METHOD FB_init : BOOL
VAR_INPUT
  /// if TRUE, the retain variables are initialized (warm start / cold start)
  bInitRetains : BOOL; 
  /// if TRUE, the instance afterwards gets moved into the copy code (online change)
  bInCopyCode  : BOOL;  
END_VAR
MyType := 'MC_CalculateInverseKinematicFB';

ExecMode := ExecutionMode.PARALLEL;
END_METHOD

METHOD PROTECTED OnCall
VAR_IN_OUT
  /// Robot assignment of function
  AxesGroup : AxesGroup; 
END_VAR
// call base implementation
SUPER^.OnCall(AxesGroup := AxesGroup);

CASE _stepCmd OF
  
  00:  IF ( _execute_R.Q )  
       THEN
         // Check function is supported and parameter are valid ?
         IF (( CheckFunctionSupported( AxesGroup := AxesGroup )) AND
             ( CheckParameterValid   ( AxesGroup := AxesGroup )))      
         THEN
           // set busy flag
           Busy := TRUE;
           // Reset command outputs
           SysDepMemSet(pDest := ADR(OutCmd), Value := 0, DataLen := SIZEOF(OutCmd));         
           // apply command parameter
          _parCmd := ParCmd;
           // init parameter sequence
          _command.ParSeq := 1;
           // create command data
           CommandData := CreateCommandPayload(AxesGroup := AxesGroup);
           // Add command to active command register
          _uniqueID := AxesGroup.Acyclic.ActiveCommandRegister.AddCmd( pCommandFB := ADR(THIS^ ));     
           // set timeout
           SetTimeout(PT := _timeoutCmd, rTimer := _timerCmd);
           // inc step counter
          _stepCmd := _stepCmd + 1;
         END_IF 
       END_IF
     

  01:  // Wait for responce received
       IF ( _responseReceived )
       THEN
         // reset response received flag
        _responseReceived := FALSE;

         CASE  _response.State 
         OF
           CmdMessageState.BUFFERED : CommandBuffered := TRUE;
           CmdMessageState.DONE     : Done            := TRUE;
           CmdMessageState.ERROR    : Error           := TRUE;
         END_CASE
                
         // Done, Aborted or Error ?
         IF (_response.State >= CmdMessageState.DONE )
         THEN
           // Reset Busy flag
           Busy := FALSE;
           // Update results
           OutCmd.JointPosition := _response.JointPosition;
           // set timeout
           SetTimeout(PT := _timeoutCmd, rTimer := _timerCmd);
           // inc step counter
          _stepCmd := _stepCmd + 1; 
         END_IF
       END_IF


  02: IF ( NOT Execute)
      THEN
        Reset();
      END_IF     

ELSE
  // invalid step
  ErrorID := RobotLibraryEvents.ERR_INVALID_STEP;
END_CASE


// Reset FB
IF ( NOT Execute )
THEN
  Reset();
END_IF
END_METHOD

METHOD INTERNAL ParseResponsePayload : DINT
VAR_INPUT
  /// Response data
  ResponseData : RobotLibraryRecvDataFB;
  /// Timestamp
  Timestamp    : SystemTime;  
END_VAR
// Table 6-639: Received CMD payload (RC to PLC) of "CalculateInverseKinematic"
// --------------------------
// Header
// --------------------------
// Byte 00 : USINT - ParSeq | State     
// Byte 01 : SINT  - AlarmMessageSeverity    
// Byte 02 : UINT  - AlarmMessageCode HB
// Byte 03 :       - AlarmMessageCode LB
// --------------------------
// Datablock
// --------------------------
// Byte 04 : REAL  - JointPosition.J1  HW HB
// Byte 05 :       - JointPosition.J1  HW LB
// Byte 06 :       - JointPosition.J1  LW HB
// Byte 07 :       - JointPosition.J1  LW LB
// Byte 08 : REAL  - JointPosition.J2  HW HB
// Byte 09 :       - JointPosition.J2 HW LB
// Byte 10 :       - JointPosition.J2  LW HB
// Byte 11 :       - JointPosition.J2  LW LB
// Byte 12 : REAL  - JointPosition.J3  HW HB
// Byte 13 :       - JointPosition.J3  HW LB
// Byte 14 :       - JointPosition.J3  LW HB
// Byte 15 :       - JointPosition.J3  LW LB
// Byte 16 : REAL  - JointPosition.J4  HW HB
// Byte 17 :       - JointPosition.J4  HW LB
// Byte 18 :       - JointPosition.J4  LW HB
// Byte 19 :       - JointPosition.J4  LW LB
// Byte 20 : REAL  - JointPosition.J5  HW HB
// Byte 21 :       - JointPosition.J5  HW LB
// Byte 22 :       - JointPosition.J5  LW HB
// Byte 23 :       - JointPosition.J5  LW LB
// Byte 24 : REAL  - JointPosition.J6  HW HB
// Byte 25 :       - JointPosition.J6  HW LB
// Byte 26 :       - JointPosition.J6  LW HB
// Byte 27 :       - JointPosition.J6  LW LB
// Byte 28 : REAL  - JointPosition.E1  HW HB
// Byte 29 :       - JointPosition.E1  HW LB
// Byte 30 :       - JointPosition.E1  LW HB
// Byte 31 :       - JointPosition.E1  LW LB
// Byte 32 : REAL  - JointPosition.E2  HW HB
// Byte 33 :       - JointPosition.E2  HW LB
// Byte 34 :       - JointPosition.E2  LW HB
// Byte 35 :       - JointPosition.E2  LW LB
// Byte 36 : REAL  - JointPosition.E3  HW HB
// Byte 37 :       - JointPosition.E3  HW LB
// Byte 38 :       - JointPosition.E3  LW HB
// Byte 39 :       - JointPosition.E3  LW LB
// Byte 40 : REAL  - JointPosition.E4  HW HB
// Byte 41 :       - JointPosition.E4  HW LB
// Byte 42 :       - JointPosition.E4  LW HB
// Byte 43 :       - JointPosition.E4  LW LB
// Byte 44 : REAL  - JointPosition.E5  HW HB
// Byte 45 :       - JointPosition.E5  HW LB
// Byte 46 :       - JointPosition.E5  LW HB
// Byte 47 :       - JointPosition.E5  LW LB
// Byte 48 : REAL  - JointPosition.E6  HW HB
// Byte 49 :       - JointPosition.E6  HW LB
// Byte 50 :       - JointPosition.E6  LW HB
// Byte 51 :       - JointPosition.E6  LW LB
// --------------------------
// call base implementation to parse the header from payload buffer
ResponseData.PayloadPtr := SUPER^.ParseResponsePayload(ResponseData := ResponseData, Timestamp := Timestamp);

// copy parsed header to response
_response.ParSeq               := _rspHeader.ParSeq;
_response.State                := _rspHeader.State;
_response.AlarmMessageSeverity := _rspHeader.AlarmMessageSeverity;
_response.AlarmMessageCode     := _rspHeader.AlarmMessageCode;

// Get Response.JointPosition.J1
_response.JointPosition.J1 := ResponseData.GetReal();
// Get Response.JointPosition.J2
_response.JointPosition.J2 := ResponseData.GetReal();
// Get Response.JointPosition.J3
_response.JointPosition.J3 := ResponseData.GetReal();
// Get Response.JointPosition.J4
_response.JointPosition.J4 := ResponseData.GetReal();
// Get Response.JointPosition.J5
_response.JointPosition.J5 := ResponseData.GetReal();
// Get Response.JointPosition.J6
_response.JointPosition.J6 := ResponseData.GetReal();
// Get Response.JointPosition.E1
_response.JointPosition.E1 := ResponseData.GetReal();
// Get Response.JointPosition.E2
_response.JointPosition.E2 := ResponseData.GetReal();
// Get Response.JointPosition.E3
_response.JointPosition.E3 := ResponseData.GetReal();
// Get Response.JointPosition.E4
_response.JointPosition.E4 := ResponseData.GetReal();
// Get Response.JointPosition.E5
_response.JointPosition.E5 := ResponseData.GetReal();
// Get Response.JointPosition.E6
_response.JointPosition.E6 := ResponseData.GetReal();

// Create logging
ParseResponsePayloadLog(ResponseData := ResponseData, Timestamp := Timestamp);
END_METHOD

METHOD INTERNAL ParseResponsePayloadLog
VAR_INPUT
  /// Response data
  ResponseData : RobotLibraryRecvDataFB;
  /// Timestamp
  Timestamp    : SystemTime;  
END_VAR
// Create log entry for Parameter start
CreateLogMessage      ( Timestamp   := Timestamp,
                        MessageType := MessageType.CMD,
                        Severity    := Severity.DEBUG,
                        MessageCode := 0,
                        MessageText := 'Parsed the following parameter(s) from response data:');
                        
// Create log entry for JointPosition.J1
CreateLogMessagePara1 ( Timestamp   := Timestamp,
                        MessageType := MessageType.CMD,
                        Severity    := Severity.DEBUG,
                        MessageCode := 0,
                        MessageText := 'Response.JointPosition.J1 = {1}',
                        Para1       :=  REAL_TO_STRING(_response.JointPosition.J1));

// Create log entry for JointPosition.J2
CreateLogMessagePara1 ( Timestamp   := Timestamp,
                        MessageType := MessageType.CMD,
                        Severity    := Severity.DEBUG,
                        MessageCode := 0,
                        MessageText := 'Response.JointPosition.J2 = {1}',
                        Para1       :=  REAL_TO_STRING(_response.JointPosition.J2));

// Create log entry for JointPosition.J3
CreateLogMessagePara1 ( Timestamp   := Timestamp,
                        MessageType := MessageType.CMD,
                        Severity    := Severity.DEBUG,
                        MessageCode := 0,
                        MessageText := 'Response.JointPosition.J3 = {1}',
                        Para1       :=  REAL_TO_STRING(_response.JointPosition.J3));

// Create log entry for JointPosition.J4
CreateLogMessagePara1 ( Timestamp   := Timestamp,
                        MessageType := MessageType.CMD,
                        Severity    := Severity.DEBUG,
                        MessageCode := 0,
                        MessageText := 'Response.JointPosition.J4 = {1}',
                        Para1       :=  REAL_TO_STRING(_response.JointPosition.J4));

// Create log entry for JointPosition.J5
CreateLogMessagePara1 ( Timestamp   := Timestamp,
                        MessageType := MessageType.CMD,
                        Severity    := Severity.DEBUG,
                        MessageCode := 0,
                        MessageText := 'Response.JointPosition.J5 = {1}',
                        Para1       :=  REAL_TO_STRING(_response.JointPosition.J5));

// Create log entry for JointPosition.J6
CreateLogMessagePara1 ( Timestamp   := Timestamp,
                        MessageType := MessageType.CMD,
                        Severity    := Severity.DEBUG,
                        MessageCode := 0,
                        MessageText := 'Response.JointPosition.J6 = {1}',
                        Para1       :=  REAL_TO_STRING(_response.JointPosition.J6));

// Create log entry for JointPosition.E1
CreateLogMessagePara1 ( Timestamp   := Timestamp,
                        MessageType := MessageType.CMD,
                        Severity    := Severity.DEBUG,
                        MessageCode := 0,
                        MessageText := 'Response.JointPosition.E1 = {1}',
                        Para1       :=  REAL_TO_STRING(_response.JointPosition.E1));

// Create log entry for JointPosition.E2
CreateLogMessagePara1 ( Timestamp   := Timestamp,
                        MessageType := MessageType.CMD,
                        Severity    := Severity.DEBUG,
                        MessageCode := 0,
                        MessageText := 'Response.JointPosition.E2 = {1}',
                        Para1       :=  REAL_TO_STRING(_response.JointPosition.E2));

// Create log entry for JointPosition.E3
CreateLogMessagePara1 ( Timestamp   := Timestamp,
                        MessageType := MessageType.CMD,
                        Severity    := Severity.DEBUG,
                        MessageCode := 0,
                        MessageText := 'Response.JointPosition.E3 = {1}',
                        Para1       :=  REAL_TO_STRING(_response.JointPosition.E3));

// Create log entry for JointPosition.E4
CreateLogMessagePara1 ( Timestamp   := Timestamp,
                        MessageType := MessageType.CMD,
                        Severity    := Severity.DEBUG,
                        MessageCode := 0,
                        MessageText := 'Response.JointPosition.E4 = {1}',
                        Para1       :=  REAL_TO_STRING(_response.JointPosition.E4));

// Create log entry for JointPosition.E5
CreateLogMessagePara1 ( Timestamp   := Timestamp,
                        MessageType := MessageType.CMD,
                        Severity    := Severity.DEBUG,
                        MessageCode := 0,
                        MessageText := 'Response.JointPosition.E5 = {1}',
                        Para1       :=  REAL_TO_STRING(_response.JointPosition.E5));

// Create log entry for JointPosition.E6
CreateLogMessagePara1 ( Timestamp   := Timestamp,
                        MessageType := MessageType.CMD,
                        Severity    := Severity.DEBUG,
                        MessageCode := 0,
                        MessageText := 'Response.JointPosition.E6 = {1}',
                        Para1       :=  REAL_TO_STRING(_response.JointPosition.E6));
END_METHOD

METHOD PROTECTED Reset : DINT
VAR_INPUT
END_VAR
Reset := SUPER^.Reset();

Done               := FALSE;
Busy               := FALSE;
CommandBuffered    := FALSE;
END_METHOD

END_FUNCTION_BLOCK

// Library/POUs/Calculation/MC_CalculateTool/MC_CalculateToolFB
/// Calculate tool (TCP) with four-point method
FUNCTION_BLOCK MC_CalculateToolFB EXTENDS RobotLibraryBaseExecuteFB
// ------------------------------------------------------------------------- 
//  SRCI Robot Library                                                
// ------------------------------------------------------------------------- 
//                                                                           
//  Object:      CalculateToolFB                                       
//  Author:      Thorsten Brach                                                
//  Date:        2024-06-09
//
//  Description:                                              
//   
//                                                                           
//  Copyright: 
//    (C) 2024 Thorsten Brach. All rights reserved                                                                                                                                            
//             Licensed under the LGPL-3.0 license.
//                                                                           
//  Disclaimer:                                                                           
//    This project is provided without any guarantee and can be used for   
//    private and commercial purposes. Any use is at the user’s 
//    own risk and responsibility.
//
// -------------------------------------------------------------------------
VAR_INPUT
  /// Command parameter 
  ParCmd          : CalculateToolParCmd;      
END_VAR
VAR_OUTPUT
  /// Command is transferred and confirmed by the RC
  CommandBuffered : BOOL;
  /// Command output 
  OutCmd          : CalculateToolOutCmd;  
END_VAR

VAR
  /// internal copy of command parameter 
 _parCmd          : CalculateToolParCmd;
  /// command data to send
 _command         : CalculateToolSendData;
  /// response data received
 _response        : CalculateToolRecvData;      
  /// Incremented with each position of the input parameter "PositionsArray" sent from the PLC to the RC.
  /// • Default: 0
 _dataIndex       : USINT;
  /// Set TRUE by the client, when according to the user selected "Mode" the final position of the input parameter "PositionsArray" is sent to the RC.
  /// • Default: FALSE
 _dataComplete    : BOOL;
END_VAR

SUPER^(AxesGroup := AxesGroup);

METHOD PROTECTED CheckFunctionSupported : BOOL
VAR_IN_OUT
  /// Robot assignment of function
  AxesGroup : AxesGroup; 
END_VAR
CheckFunctionSupported := AxesGroup.InternalData.RCSupportedFunctions.CalculateTool;

IF ( NOT CheckFunctionSupported )
THEN
  // call base implementation for set error and create log entry
  SUPER^.CheckFunctionSupported(AxesGroup := AxesGroup);
END_IF
END_METHOD

METHOD PROTECTED CheckParameterChanged : BOOL
VAR_IN_OUT
  /// Robot assignment of function
  AxesGroup    : AxesGroup; 
END_VAR
// Check ParCmd Size is > 0, because MemCmp does not work correctly with size = 0
IF (SIZEOF(ParCmd) = 0) 
THEN 
  RETURN;
END_IF

// compare memory 
_parameterChanged := ( SysDepMemCmp(pData1 := ADR(ParCmd), pData2 := ADR(_parCmd), DataLen := SIZEOF(ParCmd)) <> RobotLibraryConstants.OK );

// check parameter valid ?
_parameterValid   := CheckParameterValid( AxesGroup := AxesGroup );

IF ((  _parameterChanged        )  AND 
    (  _parameterValid          )) OR
    (  _parameterUpdateInternal )  
THEN  
  // reset internal flag for send parameter update
 _parameterUpdateInternal := FALSE;
  // update internal copy of parameters 
 _parCmd := ParCmd;
  // inc parameter sequence
 _command.ParSeq := _command.ParSeq + 1;
  // update command data  
  CommandData := CreateCommandPayload(AxesGroup := AxesGroup); // ( Access via reference to rCommandFB in ACR )
  // notify active command register 
  AxesGroup.Acyclic.ActiveCommandRegister.NotifyParameterChanged := _uniqueID;
END_IF
END_METHOD

METHOD INTERNAL CreateCommandPayload : RobotLibrarySendDataFB
VAR_IN_OUT
  /// Robot assignment of function
  AxesGroup : AxesGroup; 
END_VAR
// Table 6-650: Sent CMD payload (PLC to RC) of "CalculateTool"
// --------------------------
// Header
// --------------------------
// Byte 00 : UINT       - Type HB     
// Byte 01 :            - Type LB    
// Byte 02 : USINT      - Reserve | ExecutionMode
// Byte 03 : USINT      - ParSeq  | Priority
// --------------------------
// Datablock
// --------------------------
// Byte 04 : USINT      - DataIndex
// Byte 05 : BOOL       - DataComplete
// Byte 06 : USINT      - ToolNo
// Byte 07 : USINT      - FrameNo
// Byte 08 : SINT       - Mode
// Byte 09 : USINT      - ExternalTCP
// Byte 10 : REAL       - Position.X  HW HB
// Byte 11 :            - Position.X  HW LB
// Byte 12 :            - Position.X  LW HB
// Byte 13 :            - Position.X  LW LB
// Byte 14 : REAL       - Position.Y  HW HB
// Byte 15 :            - Position.Y  HW LB
// Byte 16 :            - Position.Y  LW HB
// Byte 17 :            - Position.Y  LW LB
// Byte 18 : REAL       - Position.Z  HW HB
// Byte 19 :            - Position.Z  HW LB
// Byte 20 :            - Position.Z  LW HB
// Byte 21 :            - Position.Z  LW LB
// Byte 22 : REAL       - Position.Rx HW HB
// Byte 23 :            - Position.Rx HW LB
// Byte 24 :            - Position.Rx LW HB
// Byte 25 :            - Position.Rx LW LB
// Byte 26 : REAL       - Position.Ry HW HB
// Byte 27 :            - Position.Ry HW LB
// Byte 28 :            - Position.Ry LW HB
// Byte 29 :            - Position.Ry LW LB
// Byte 30 : REAL       - Position.Rz HW HB
// Byte 31 :            - Position.Rz HW LB
// Byte 32 :            - Position.Rz LW HB
// Byte 33 :            - Position.Rz LW LB
// Byte 34 : Config     - ArmConfig   LW HB
// Byte 35 :            - ArmConfig   LW LB
// Byte 36 : TurnNumber - J1 + J2     LW HB
// Byte 37 :            - J3 + J4     LW LB
// Byte 38 :            - J5 + J6     LW LB
// Byte 39 :            - E1          LW LB
// Byte 40 : REAL       - Position.E1 HW HB
// Byte 41 :            - Position.E1 HW LB
// Byte 42 :            - Position.E1 LW HB
// Byte 43 :            - Position.E1 LW LB
// Byte 44 : REAL       - Position.E2 HW HB
// Byte 45 :            - Position.E2 HW LB
// Byte 46 :            - Position.E2 LW HB
// Byte 47 :            - Position.E2 LW LB
// Byte 48 : REAL       - Position.E3 HW HB
// Byte 49 :            - Position.E3 HW LB
// Byte 50 :            - Position.E3 LW HB
// Byte 51 :            - Position.E3 LW LB
// Byte 52 : REAL       - Position.E4 HW HB
// Byte 53 :            - Position.E4 HW LB
// Byte 54 :            - Position.E4 LW HB
// Byte 55 :            - Position.E4 LW LB
// Byte 56 : REAL       - Position.E5 HW HB
// Byte 57 :            - Position.E5 HW LB
// Byte 58 :            - Position.E5 LW HB
// Byte 59 :            - Position.E5 LW LB
// Byte 60 : REAL       - Position.E6 HW HB
// Byte 61 :            - Position.E6 HW LB
// Byte 62 :            - Position.E6 LW HB
// Byte 63 :            - Position.E6 LW LB
// --------------------------
// set command parameter 
_command.CmdTyp         :=  CmdType.CalculateTool;
_command.ExecMode       :=  ExecMode;
_command.ParSeq         := _command.ParSeq;
_command.Priority       :=  Priority;
_command.DataIndex      := _dataIndex;
_command.DataComplete.0 := _dataComplete;
_command.ToolNo         := _parCmd.ToolNo;
_command.FrameNo        := _parCmd.FrameNo;
_command.Mode           := _parCmd.Mode;
_command.ExternalTCP.0  := _parCmd.ExternalTCP;
  
// copy command data to header
_cmdHeader := _command;
// call base implementation to copy header to payload buffer
CreateCommandPayload := SUPER^.CreateCommandPayload(AxesGroup := AxesGroup);

// add command.TargetFrameNo
CreateCommandPayload.AddUsint(_command.DataIndex);
// add command.DataComplete
CreateCommandPayload.AddByte(_command.DataComplete);
// add command.ToolNo
CreateCommandPayload.AddUsint(_command.ToolNo);
// add command.FrameNo
CreateCommandPayload.AddUsint(_command.FrameNo);
// add command.Mode
CreateCommandPayload.AddSint(_command.Mode);
// add command.Mode
CreateCommandPayload.AddUsint(_command.ExternalTCP);
// add command.Position.X
CreateCommandPayload.AddReal(_command.Position.X);
// add command.Position.Y
CreateCommandPayload.AddReal(_command.Position.Y);
// add command.Position.Z
CreateCommandPayload.AddReal(_command.Position.Z);
// add command.Position.Rx
CreateCommandPayload.AddReal(_command.Position.Rx);
// add command.Position.Ry
CreateCommandPayload.AddReal(_command.Position.Ry);
// add command.Position.Rz
CreateCommandPayload.AddReal(_command.Position.Rz);
// add command.Position.Config
CreateCommandPayload.AddArmConfig (_command.Position.Config);
// add command.Position.TurnNumber
CreateCommandPayload.AddTurnNumber(_command.Position.TurnNumber);
// add command.Position.E1
CreateCommandPayload.AddReal(_command.Position.E1);
// add command.Position.E2
CreateCommandPayload.AddReal(_command.Position.E2);
// add command.Position.E3
CreateCommandPayload.AddReal(_command.Position.E3);
// add command.Position.E4
CreateCommandPayload.AddReal(_command.Position.E4);
// add command.Position.E5
CreateCommandPayload.AddReal(_command.Position.E5);
// add command.Position.E6
CreateCommandPayload.AddReal(_command.Position.E6);

// Create logging
CreateCommandPayloadLog(AxesGroup := AxesGroup);
END_METHOD

METHOD INTERNAL CreateCommandPayloadLog 
VAR_IN_OUT
  /// Robot assignment of function
  AxesGroup : AxesGroup; 
END_VAR
// Create log entry for Parameter start
CreateLogMessage      ( Timestamp   := AxesGroup.InternalData.SystemTime,
                        MessageType := MessageType.CMD,
                        Severity    := Severity.DEBUG,
                        MessageCode := 0,
                        MessageText := 'Create command payload with the following parameter(s) :');

// Create log entry for DataIndex
CreateLogMessagePara1 ( Timestamp   := AxesGroup.InternalData.SystemTime,
                        MessageType := MessageType.CMD,
                        Severity    := Severity.DEBUG,
                        MessageCode := 0,
                        MessageText := 'Command.DataIndex = {1}',
                        Para1       :=  USINT_TO_STRING(_command.DataIndex));

// Create log entry for DataComplete
CreateLogMessagePara1 ( Timestamp   := AxesGroup.InternalData.SystemTime,
                        MessageType := MessageType.CMD,
                        Severity    := Severity.DEBUG,
                        MessageCode := 0,
                        MessageText := 'Command.DataComplete = {1}',
                        Para1       :=  BYTE_TO_STRING(_command.DataComplete));

// Create log entry for ToolNo
CreateLogMessagePara1 ( Timestamp   := AxesGroup.InternalData.SystemTime,
                        MessageType := MessageType.CMD,
                        Severity    := Severity.DEBUG,
                        MessageCode := 0,
                        MessageText := 'Command.ToolNo = {1}',
                        Para1       :=  USINT_TO_STRING(_command.ToolNo));

// Create log entry for FrameNo
CreateLogMessagePara1 ( Timestamp   := AxesGroup.InternalData.SystemTime,
                        MessageType := MessageType.CMD,
                        Severity    := Severity.DEBUG,
                        MessageCode := 0,
                        MessageText := 'Command.FrameNo = {1}',
                        Para1       :=  USINT_TO_STRING(_command.FrameNo));

// Create log entry for Mode
CreateLogMessagePara1 ( Timestamp   := AxesGroup.InternalData.SystemTime,
                        MessageType := MessageType.CMD,
                        Severity    := Severity.DEBUG,
                        MessageCode := 0,
                        MessageText := 'Command.Mode = {1}',
                        Para1       :=  TOOL_CALCULATION_MODE_TO_STRING(_command.Mode));

// Create log entry for ExternalTCP
CreateLogMessagePara1 ( Timestamp   := AxesGroup.InternalData.SystemTime,
                        MessageType := MessageType.CMD,
                        Severity    := Severity.DEBUG,
                        MessageCode := 0,
                        MessageText := 'Command.ExternalTCP = {1}',
                        Para1       :=  BOOL_TO_STRING(_command.ExternalTCP.0));

// Create log entry for Position.X
CreateLogMessagePara1 ( Timestamp   := AxesGroup.InternalData.SystemTime,
                        MessageType := MessageType.CMD,
                        Severity    := Severity.DEBUG,
                        MessageCode := 0,
                        MessageText := 'Command.Position.X = {1}',
                        Para1       :=  REAL_TO_STRING(_command.Position.X));

// Create log entry for Position.Y
CreateLogMessagePara1 ( Timestamp   := AxesGroup.InternalData.SystemTime,
                        MessageType := MessageType.CMD,
                        Severity    := Severity.DEBUG,
                        MessageCode := 0,
                        MessageText := 'Command.Position.Y = {1}',
                        Para1       :=  REAL_TO_STRING(_command.Position.Y));

// Create log entry for Position.Z
CreateLogMessagePara1 ( Timestamp   := AxesGroup.InternalData.SystemTime,
                        MessageType := MessageType.CMD,
                        Severity    := Severity.DEBUG,
                        MessageCode := 0,
                        MessageText := 'Command.Position.Z = {1}',
                        Para1       :=  REAL_TO_STRING(_command.Position.Z));

// Create log entry for Position.Rx
CreateLogMessagePara1 ( Timestamp   := AxesGroup.InternalData.SystemTime,
                        MessageType := MessageType.CMD,
                        Severity    := Severity.DEBUG,
                        MessageCode := 0,
                        MessageText := 'Command.Position.Rx = {1}',
                        Para1       :=  REAL_TO_STRING(_command.Position.Rx));

// Create log entry for Position.Ry
CreateLogMessagePara1 ( Timestamp   := AxesGroup.InternalData.SystemTime,
                        MessageType := MessageType.CMD,
                        Severity    := Severity.DEBUG,
                        MessageCode := 0,
                        MessageText := 'Command.Position.Ry = {1}',
                        Para1       :=  REAL_TO_STRING(_command.Position.Ry));

// Create log entry for Position.Rz
CreateLogMessagePara1 ( Timestamp   := AxesGroup.InternalData.SystemTime,
                        MessageType := MessageType.CMD,
                        Severity    := Severity.DEBUG,
                        MessageCode := 0,
                        MessageText := 'Command.Position.Rz = {1}',
                        Para1       :=  REAL_TO_STRING(_command.Position.Rz));

// Create log entry for Position.Config
CreateLogMessagePara1 ( Timestamp   := AxesGroup.InternalData.SystemTime,
                        MessageType := MessageType.CMD,
                        Severity    := Severity.DEBUG,
                        MessageCode := 0,
                        MessageText := 'Command.Position.Config = {1}',
                        Para1       :=  ARM_CONFIG_TO_STRING(_command.Position.Config));

// Create log entry for Position.TurnNumber[0]
CreateLogMessagePara1 ( Timestamp   := AxesGroup.InternalData.SystemTime,
                        MessageType := MessageType.CMD,
                        Severity    := Severity.DEBUG,
                        MessageCode := 0,
                        MessageText := 'Command.Position.TurnNumber[0] = {1}',
                        Para1       :=  BYTE_TO_STRING(CombineHalfSints(HalfSintHi := _command.Position.TurnNumber.J2Turns, 
                                                                        HalfSintLo := _command.Position.TurnNumber.J1Turns)));

// Create log entry for Position.TurnNumber[1]
CreateLogMessagePara1 ( Timestamp   := AxesGroup.InternalData.SystemTime,
                        MessageType := MessageType.CMD,
                        Severity    := Severity.DEBUG,
                        MessageCode := 0,
                        MessageText := 'Command.Position.TurnNumber[1] = {1}',
                        Para1       :=  BYTE_TO_STRING(CombineHalfSints(HalfSintHi := _command.Position.TurnNumber.J4Turns, 
                                                                        HalfSintLo := _command.Position.TurnNumber.J3Turns)));

// Create log entry for Position.TurnNumber[2]
CreateLogMessagePara1 ( Timestamp   := AxesGroup.InternalData.SystemTime,
                        MessageType := MessageType.CMD,
                        Severity    := Severity.DEBUG,
                        MessageCode := 0,
                        MessageText := 'Command.Position.TurnNumber[2] = {1}',
                        Para1       :=  BYTE_TO_STRING(CombineHalfSints(HalfSintHi := _command.Position.TurnNumber.J6Turns, 
                                                                        HalfSintLo := _command.Position.TurnNumber.J5Turns)));

// Create log entry for Position.TurnNumber[3]
CreateLogMessagePara1 ( Timestamp   := AxesGroup.InternalData.SystemTime,
                        MessageType := MessageType.CMD,
                        Severity    := Severity.DEBUG,
                        MessageCode := 0,
                        MessageText := 'Command.Position.TurnNumber[3] = {1}',
                        Para1       :=  SINT_TO_STRING(_command.Position.TurnNumber.E1Turns));

// Create log entry for Position.E1
CreateLogMessagePara1 ( Timestamp   := AxesGroup.InternalData.SystemTime,
                        MessageType := MessageType.CMD,
                        Severity    := Severity.DEBUG,
                        MessageCode := 0,
                        MessageText := 'Command.Position.E1 = {1}',
                        Para1       :=  REAL_TO_STRING(_command.Position.E1));

// Create log entry for Position.E2
CreateLogMessagePara1 ( Timestamp   := AxesGroup.InternalData.SystemTime,
                        MessageType := MessageType.CMD,
                        Severity    := Severity.DEBUG,
                        MessageCode := 0,
                        MessageText := 'Command.Position.E2 = {1}',
                        Para1       :=  REAL_TO_STRING(_command.Position.E2));

// Create log entry for Position.E3
CreateLogMessagePara1 ( Timestamp   := AxesGroup.InternalData.SystemTime,
                        MessageType := MessageType.CMD,
                        Severity    := Severity.DEBUG,
                        MessageCode := 0,
                        MessageText := 'Command.Position.E3 = {1}',
                        Para1       :=  REAL_TO_STRING(_command.Position.E3));

// Create log entry for Position.E4
CreateLogMessagePara1 ( Timestamp   := AxesGroup.InternalData.SystemTime,
                        MessageType := MessageType.CMD,
                        Severity    := Severity.DEBUG,
                        MessageCode := 0,
                        MessageText := 'Command.Position.E4 = {1}',
                        Para1       :=  REAL_TO_STRING(_command.Position.E4));

// Create log entry for Position.E5
CreateLogMessagePara1 ( Timestamp   := AxesGroup.InternalData.SystemTime,
                        MessageType := MessageType.CMD,
                        Severity    := Severity.DEBUG,
                        MessageCode := 0,
                        MessageText := 'Command.Position.E5 = {1}',
                        Para1       :=  REAL_TO_STRING(_command.Position.E5));

// Create log entry for Position.E6
CreateLogMessagePara1 ( Timestamp   := AxesGroup.InternalData.SystemTime,
                        MessageType := MessageType.CMD,
                        Severity    := Severity.DEBUG,
                        MessageCode := 0,
                        MessageText := 'Command.Position.E6 = {1}',
                        Para1       :=  REAL_TO_STRING(_command.Position.E6));
END_METHOD

METHOD FB_init : BOOL
VAR_INPUT
  /// if TRUE, the retain variables are initialized (warm start / cold start)
  bInitRetains : BOOL; 
  /// if TRUE, the instance afterwards gets moved into the copy code (online change)
  bInCopyCode  : BOOL;  
END_VAR
MyType := 'MC_CalculateToolFB';

ExecMode := ExecutionMode.PARALLEL;
END_METHOD

METHOD PROTECTED OnCall
VAR_IN_OUT
  /// Robot assignment of function
  AxesGroup : AxesGroup; 
END_VAR
// call base implementation
SUPER^.OnCall(AxesGroup := AxesGroup);

CASE _stepCmd OF
  
  00:  IF ( _execute_R.Q )  
       THEN
         // Check function is supported and parameter are valid ?
         IF (( CheckFunctionSupported( AxesGroup := AxesGroup )) AND
             ( CheckParameterValid   ( AxesGroup := AxesGroup )))      
         THEN
           // set busy flag
           Busy := TRUE;
           // Reset command outputs
           SysDepMemSet(pDest := ADR(OutCmd), Value := 0, DataLen := SIZEOF(OutCmd));         
           // apply command parameter
          _parCmd := ParCmd;
           // init parameter sequence
          _command.ParSeq := 1;
           // set timeout
           SetTimeout(PT := _timeoutCmd, rTimer := _timerCmd);
           // inc step counter
          _stepCmd := _stepCmd + 1;
         END_IF 
       END_IF
     

  01: // inc data index 
     _dataIndex := _dataIndex + 1;

      CASE _parCmd.Mode OF

        ToolCalculationMode.TWO_POINT_Z_METHOD :
          _dataComplete := _dataIndex >= 2;
        
        ToolCalculationMode.THREE_POINT_METHOD :
          _dataComplete := _dataIndex >= 3;

        ToolCalculationMode.FOUR_POINT_METHOD :
          _dataComplete := _dataIndex >= 4;        

        ToolCalculationMode.FIVE_POINT_METHOD :        
          _dataComplete := _dataIndex >= 5;

        ToolCalculationMode.SIX_POINT_METHOD :        
          _dataComplete := _dataIndex >= 6;

        ToolCalculationMode.ABC_WORLD_METHOD :
          _dataComplete := _dataIndex >= 1;
        
        ToolCalculationMode.ABC_TWO_POINT_METHOD :
          _dataComplete := _dataIndex >= 2;

      END_CASE

       // create command data
       CommandData := CreateCommandPayload(AxesGroup := AxesGroup);
       // Add command to active command register
      _uniqueID := AxesGroup.Acyclic.ActiveCommandRegister.AddCmd( pCommandFB := ADR(THIS^ ));     
       // set timeout
       SetTimeout(PT := _timeoutCmd, rTimer := _timerCmd);
       // inc step counter
      _stepCmd := _stepCmd + 1; 


  02:  // Wait for responce received
       IF ( _responseReceived )
       THEN
         // reset response received flag
        _responseReceived := FALSE;

         CASE  _response.State 
         OF
           CmdMessageState.BUFFERED : CommandBuffered := TRUE;
           CmdMessageState.DONE     : Done            := TRUE;
           CmdMessageState.ERROR    : Error           := TRUE;
         END_CASE
                
         // Done, Aborted or Error ?
         IF (_response.State >= CmdMessageState.DONE )
         THEN
           // Reset Busy flag
           Busy := FALSE;
           // Update results
           OutCmd.TCPMaxError    := _response.TCPMaxError;
           OutCmd.TCPMeanError   := _response.TCPMeanError;
           OutCmd.ToolData       := _response.ToolData;
           
           IF ( _dataComplete ) OR (_response.State = CmdMessageState.ABORTED )
           THEN
             // set timeout
             SetTimeout(PT := _timeoutCmd, rTimer := _timerCmd);
             // inc step counter
            _stepCmd := _stepCmd + 1; 
           ELSE
             // set timeout
             SetTimeout(PT := _timeoutCmd, rTimer := _timerCmd);
             // dec step counter
            _stepCmd := _stepCmd - 1; 
           END_IF
         END_IF
       END_IF


  03: IF ( NOT Execute)
      THEN
        Reset(); 
      END_IF     
      
ELSE
  // invalid step
  ErrorID := RobotLibraryEvents.ERR_INVALID_STEP;
END_CASE


// Reset FB
IF ( NOT Execute )
THEN
  Reset();
END_IF
END_METHOD

METHOD INTERNAL ParseResponsePayload : DINT
VAR_INPUT
  /// Response data
  ResponseData : RobotLibraryRecvDataFB;
  /// Timestamp
  Timestamp    : SystemTime;  
END_VAR
// Table 6-651: Received CMD payload (RC to PLC) of "CalculateTool"
// --------------------------
// Header
// --------------------------
// Byte 00 : USINT      - ParSeq | State     
// Byte 01 : SINT       - AlarmMessageSeverity    
// Byte 02 : UINT       - AlarmMessageCode HB
// Byte 03 :            - AlarmMessageCode LB
// --------------------------
// Datablock
// --------------------------
// Byte 04 : IEC_DATE   - ToolData.Date LW HB
// Byte 05 :            - ToolData.Date LW LB
// Byte 06 : REAL       - TCPMaxError   HW HB
// Byte 07 :            - TCPMaxError   HW LB
// Byte 08 :            - TCPMaxError   LW HB
// Byte 09 :            - TCPMaxError   LW LB
// Byte 10 : REAL       - TCPMeanError  HW HB
// Byte 11 :            - TCPMeanError  HW LB
// Byte 12 :            - TCPMeanError  LW HB
// Byte 13 :            - TCPMeanError  LW LB
// Byte 14 : IEC_TIME   - ToolData.Time HW HB
// Byte 15 :            - ToolData.Time HW LB
// Byte 16 :            - ToolData.Time LW HB
// Byte 17 :            - ToolData.Time LW LB


// Byte 18 : REAL       - ToolData.X  HW HB
// Byte 19 :            - ToolData.X  HW LB
// Byte 20 :            - ToolData.X  LW HB
// Byte 21 :            - ToolData.X  LW LB
// Byte 22 : REAL       - ToolData.Y  HW HB
// Byte 23 :            - ToolData.Y  HW LB
// Byte 24 :            - ToolData.Y  LW HB
// Byte 25 :            - ToolData.Y  LW LB
// Byte 26 : REAL       - ToolData.Z  HW HB
// Byte 27 :            - ToolData.Z  HW LB
// Byte 28 :            - ToolData.Z  LW HB
// Byte 29 :            - ToolData.Z  LW LB
// Byte 30 : REAL       - ToolData.Rx HW HB
// Byte 31 :            - ToolData.Rx HW LB
// Byte 32 :            - ToolData.Rx LW HB
// Byte 33 :            - ToolData.Rx LW LB
// Byte 34 : REAL       - ToolData.Ry HW HB
// Byte 35 :            - ToolData.Ry HW LB
// Byte 36 :            - ToolData.Ry LW HB
// Byte 37 :            - ToolData.Ry LW LB
// Byte 38 : REAL       - ToolData.Rz HW HB
// Byte 39 :            - ToolData.Rz HW LB
// Byte 40 :            - ToolData.Rz LW HB
// Byte 41 :            - ToolData.Rz LW LB
// Byte 42 : USINT      - ToolData.ID
// Byte 43 : USINT      - ToolData.LoadNo
// Byte 44 : BOOL       - ToolData.ExternalTCP
// --------------------------
// call base implementation to parse the header from payload buffer
ResponseData.PayloadPtr := SUPER^.ParseResponsePayload(ResponseData := ResponseData, Timestamp := Timestamp);

// copy parsed header to response
_response.ParSeq                := _rspHeader.ParSeq;
_response.State                 := _rspHeader.State;
_response.AlarmMessageSeverity  := _rspHeader.AlarmMessageSeverity;
_response.AlarmMessageCode      := _rspHeader.AlarmMessageCode;

// Get Response.IEC_Date
_response.ToolData.Timestamp.IEC_Date := ResponseData.GetIecDate();
// Get Response.TCPMaxError
_response.TCPMaxError := ResponseData.GetReal();
// Get Response.TCPMeanError
_response.TCPMeanError := ResponseData.GetReal();
// Get Response.ToolData.Time
_response.ToolData.Timestamp.IEC_Time := ResponseData.GetIecTime();
// Get Response.ToolData.X
_response.ToolData.X := ResponseData.GetReal();
// Get Response.ToolData.Y            
_response.ToolData.Y := ResponseData.GetReal();
// Get Response.ToolData.Z            
_response.ToolData.Z := ResponseData.GetReal();
// Get Response.ToolData.Rx           
_response.ToolData.Rx := ResponseData.GetReal();
// Get Response.ToolData.Ry           
_response.ToolData.Ry := ResponseData.GetReal();
// Get Response.ToolData.Rz           
_response.ToolData.Rz := ResponseData.GetReal();
// Get Response.ToolData.ID           
_response.ToolData.ID := ResponseData.GetUsint();
// Get Response.ToolData.LoadNo       
_response.ToolData.LoadNo := ResponseData.GetUsint();
// Get Response.ToolData.ExternalTCP
_response.ToolData.ExternalTCP := ResponseData.GetBool();

// Create logging
ParseResponsePayloadLog(ResponseData := ResponseData, Timestamp := Timestamp);
END_METHOD

METHOD INTERNAL ParseResponsePayloadLog
VAR_INPUT
  /// Response data
  ResponseData : RobotLibraryRecvDataFB;
  /// Timestamp
  Timestamp    : SystemTime;  
END_VAR
// Create log entry for Parameter start
CreateLogMessage      ( Timestamp   := Timestamp,
                        MessageType := MessageType.CMD,
                        Severity    := Severity.DEBUG,
                        MessageCode := 0,
                        MessageText := 'Parsed the following parameter(s) from response data:');
                        
// Create log entry for IEC_Date
CreateLogMessagePara1 ( Timestamp   := Timestamp,
                        MessageType := MessageType.CMD,
                        Severity    := Severity.DEBUG,
                        MessageCode := 0,
                        MessageText := 'Response.ToolData.Timestamp.IEC_DATE = {1}',
                        Para1       :=  IEC_DATE_TO_STRING(_response.ToolData.Timestamp.IEC_DATE));

// Create log entry for TCPMaxError
CreateLogMessagePara1 ( Timestamp   := Timestamp,
                        MessageType := MessageType.CMD,
                        Severity    := Severity.DEBUG,
                        MessageCode := 0,
                        MessageText := 'Response.TCPMaxError = {1}',
                        Para1       :=  REAL_TO_STRING(_response.TCPMaxError));

// Create log entry for TCPMeanError
CreateLogMessagePara1 ( Timestamp   := Timestamp,
                        MessageType := MessageType.CMD,
                        Severity    := Severity.DEBUG,
                        MessageCode := 0,
                        MessageText := 'Response.TCPMeanError = {1}',
                        Para1       :=  REAL_TO_STRING(_response.TCPMeanError));

// Create log entry for IEC_Time
CreateLogMessagePara1 ( Timestamp   := Timestamp,
                        MessageType := MessageType.CMD,
                        Severity    := Severity.DEBUG,
                        MessageCode := 0,
                        MessageText := 'Response.ToolData.Timestamp.IEC_TIME = {1}',
                        Para1       :=  IEC_TIME_TO_STRING(_response.ToolData.Timestamp.IEC_TIME));

// Create log entry for ToolData.X
CreateLogMessagePara1 ( Timestamp   := Timestamp,
                        MessageType := MessageType.CMD,
                        Severity    := Severity.DEBUG,
                        MessageCode := 0,
                        MessageText := 'Response.ToolData.X = {1}',
                        Para1       :=  REAL_TO_STRING(_response.ToolData.X));

// Create log entry for ToolData.Y
CreateLogMessagePara1 ( Timestamp   := Timestamp,
                        MessageType := MessageType.CMD,
                        Severity    := Severity.DEBUG,
                        MessageCode := 0,
                        MessageText := 'Response.ToolData.Y = {1}',
                        Para1       :=  REAL_TO_STRING(_response.ToolData.Y));

// Create log entry for ToolData.Z
CreateLogMessagePara1 ( Timestamp   := Timestamp,
                        MessageType := MessageType.CMD,
                        Severity    := Severity.DEBUG,
                        MessageCode := 0,
                        MessageText := 'Response.ToolData.Z = {1}',
                        Para1       :=  REAL_TO_STRING(_response.ToolData.Z));

// Create log entry for ToolData.Rx
CreateLogMessagePara1 ( Timestamp   := Timestamp,
                        MessageType := MessageType.CMD,
                        Severity    := Severity.DEBUG,
                        MessageCode := 0,
                        MessageText := 'Response.ToolData.Rx = {1}',
                        Para1       :=  REAL_TO_STRING(_response.ToolData.Rx));

// Create log entry for ToolData.Ry
CreateLogMessagePara1 ( Timestamp   := Timestamp,
                        MessageType := MessageType.CMD,
                        Severity    := Severity.DEBUG,
                        MessageCode := 0,
                        MessageText := 'Response.ToolData.Ry = {1}',
                        Para1       :=  REAL_TO_STRING(_response.ToolData.Ry));

// Create log entry for ToolData.Rz
CreateLogMessagePara1 ( Timestamp   := Timestamp,
                        MessageType := MessageType.CMD,
                        Severity    := Severity.DEBUG,
                        MessageCode := 0,
                        MessageText := 'Response.ToolData.Rz = {1}',
                        Para1       :=  REAL_TO_STRING(_response.ToolData.Rz));

// Create log entry for ToolData.ID
CreateLogMessagePara1 ( Timestamp   := Timestamp,
                        MessageType := MessageType.CMD,
                        Severity    := Severity.DEBUG,
                        MessageCode := 0,
                        MessageText := 'Response.ToolData.ID = {1}',
                        Para1       :=  USINT_TO_STRING(_response.ToolData.ID));

// Create log entry for ToolData.LoadNo
CreateLogMessagePara1 ( Timestamp   := Timestamp,
                        MessageType := MessageType.CMD,
                        Severity    := Severity.DEBUG,
                        MessageCode := 0,
                        MessageText := 'Response.ToolData.LoadNo = {1}',
                        Para1       :=  USINT_TO_STRING(_response.ToolData.LoadNo));

// Create log entry for ToolData.ExternalTCP
CreateLogMessagePara1 ( Timestamp   := Timestamp,
                        MessageType := MessageType.CMD,
                        Severity    := Severity.DEBUG,
                        MessageCode := 0,
                        MessageText := 'Response.ToolData.ExternalTCP = {1}',
                        Para1       :=  BOOL_TO_STRING(_response.ToolData.ExternalTCP));
END_METHOD

METHOD PROTECTED Reset : DINT
VAR_INPUT
END_VAR
Reset := SUPER^.Reset();

Done               := FALSE;
Busy               := FALSE;
CommandBuffered    := FALSE;
END_METHOD

END_FUNCTION_BLOCK

// Library/POUs/Calculation/MC_LoadMeasurementAutomatic/MC_LoadMeasurementAutomaticFB
/// Automatic detection of load data
FUNCTION_BLOCK MC_LoadMeasurementAutomaticFB EXTENDS RobotLibraryBaseExecuteFB
// ------------------------------------------------------------------------- 
//  SRCI Robot Library                                                
// ------------------------------------------------------------------------- 
//                                                                           
//  Object:      LoadMeasurementAutomaticFB                                       
//  Author:      Thorsten Brach                                                
//  Date:        2024-06-01
//
//  Description:                                              
//   
//                                                                           
//  Copyright: 
//    (C) 2024 Thorsten Brach. All rights reserved                                                                                                                                            
//             Licensed under the LGPL-3.0 license.
//                                                                           
//  Disclaimer:                                                                           
//    This project is provided without any guarantee and can be used for   
//    private and commercial purposes. Any use is at the user’s 
//    own risk and responsibility.
//
// -------------------------------------------------------------------------
VAR_INPUT
  /// Parameter which determines the behavior towards the previously sent and still active or buffered commands.
  AbortingMode    : AbortingMode;
  /// Defines the target sequence in which the command will be executed
  SequenceFlag    : SequenceFlag;  
  /// Command parameter 
  ParCmd          : LoadMeasurementAutomaticParCmd;      
END_VAR

VAR_OUTPUT
  /// Command is transferred and confirmed by the RC
  CommandBuffered    : BOOL;  
  /// The command takes control of the motion of the according axis group.
  Active             : BOOL;
  /// The command was aborted by another command.
  CommandAborted     : BOOL;
  /// TRUE, while command is interrupted during execution and can be continued.
  CommandInterrupted : BOOL;
  /// Command output 
  OutCmd             : LoadMeasurementAutomaticOutCmd;        
END_VAR

VAR
  /// internal copy of command parameter 
 _parCmd          : LoadMeasurementAutomaticParCmd;
  /// command data to send
 _command         : LoadMeasurementAutomaticSendData;
  /// response data received
 _response        : LoadMeasurementAutomaticRecvData;      
END_VAR

SUPER^(AxesGroup := AxesGroup);

METHOD PROTECTED CheckFunctionSupported : BOOL
VAR_IN_OUT
  /// Robot assignment of function
  AxesGroup : AxesGroup; 
END_VAR
CheckFunctionSupported := AxesGroup.InternalData.RCSupportedFunctions.LoadMeasurementAutomatic;

IF ( NOT CheckFunctionSupported )
THEN
  // call base implementation for set error and create log entry
  SUPER^.CheckFunctionSupported(AxesGroup := AxesGroup);
END_IF
END_METHOD

METHOD PROTECTED CheckParameterChanged : BOOL
VAR_IN_OUT
  /// Robot assignment of function
  AxesGroup    : AxesGroup; 
END_VAR
// Check ParCmd Size is > 0, because MemCmp does not work correctly with size = 0
IF (SIZEOF(ParCmd) = 0) 
THEN 
  RETURN;
END_IF

// compare memory 
_parameterChanged := ( SysDepMemCmp(pData1 := ADR(ParCmd), pData2 := ADR(_parCmd), DataLen := SIZEOF(ParCmd)) <> RobotLibraryConstants.OK );

// check parameter valid ?
_parameterValid   := CheckParameterValid( AxesGroup := AxesGroup );

IF ((  _parameterChanged        )  AND 
    (  _parameterValid          )) OR
    (  _parameterUpdateInternal )  
THEN  
  // reset internal flag for send parameter update
 _parameterUpdateInternal := FALSE;
  // update internal copy of parameters 
 _parCmd := ParCmd;
  // inc parameter sequence
 _command.ParSeq := _command.ParSeq + 1;
  // update command data  
  CommandData := CreateCommandPayload(AxesGroup := AxesGroup); // ( Access via reference to rCommandFB in ACR )
  // notify active command register 
  AxesGroup.Acyclic.ActiveCommandRegister.NotifyParameterChanged := _uniqueID;
END_IF
END_METHOD

METHOD INTERNAL CreateCommandPayload : RobotLibrarySendDataFB
VAR_IN_OUT
  /// Robot assignment of function
  AxesGroup : AxesGroup; 
END_VAR
// Table 6-778: Sent CMD payload (PLC to RC) of "LoadMeasurementAutomatic"
// --------------------------
// Header
// --------------------------
// Byte 000 : UINT  - Type HB     
// Byte 001 :       - Type LB    
// Byte 002 : USINT - Reserve | ExecutionMode
// Byte 003 : USINT - ParSeq  | Priority
// --------------------------
// Datablock
// --------------------------
// Byte 004 : REAL       - Mass HW HB
// Byte 005 :            - Mass HW LB
// Byte 006 :            - Mass LW HB
// Byte 007 :            - Mass LW LB
// Byte 008 : USINT      - Mode
// Byte 009 : BYTE       - Reserved
// Byte 010 : REAL       - AreaJ3[0] HW HB
// Byte 011 :            - AreaJ3[0] HW LB
// Byte 012 :            - AreaJ3[0] LW HB
// Byte 013 :            - AreaJ3[0] LW LB
// Byte 014 : REAL       - AreaJ3[1] HW HB
// Byte 015 :            - AreaJ3[1] HW LB
// Byte 016 :            - AreaJ3[1] LW HB
// Byte 017 :            - AreaJ3[1] LW LB
// Byte 018 : REAL       - AreaJ4[0] HW HB
// Byte 019 :            - AreaJ4[0] HW LB
// Byte 020 :            - AreaJ4[0] LW HB
// Byte 021 :            - AreaJ4[0] LW LB
// Byte 022 : REAL       - AreaJ4[1] HW HB
// Byte 023 :            - AreaJ4[1] HW LB
// Byte 024 :            - AreaJ4[1] LW HB
// Byte 025 :            - AreaJ4[1] LW LB
// Byte 026 : REAL       - AreaJ5[0] HW HB
// Byte 027 :            - AreaJ5[0] HW LB
// Byte 028 :            - AreaJ5[0] LW HB
// Byte 029 :            - AreaJ5[0] LW LB
// Byte 030 : REAL       - AreaJ5[1] HW HB
// Byte 031 :            - AreaJ5[1] HW LB
// Byte 032 :            - AreaJ5[1] LW HB
// Byte 033 :            - AreaJ5[1] LW LB
// Byte 034 : REAL       - AreaJ6[0] HW HB
// Byte 035 :            - AreaJ6[0] HW LB
// Byte 036 :            - AreaJ6[0] LW HB
// Byte 037 :            - AreaJ6[0] LW LB
// Byte 038 : REAL       - AreaJ6[1] HW HB
// Byte 039 :            - AreaJ6[1] HW LB
// Byte 040 :            - AreaJ6[1] LW HB
// Byte 041 :            - AreaJ6[1] LW LB
// Byte 042 : REAL       - ConfigurationAngle HW HB
// Byte 043 :            - ConfigurationAngle HW LB
// Byte 044 :            - ConfigurationAngle LW HB
// Byte 045 :            - ConfigurationAngle LW LB
// Byte 046 : REAL       - Position_1.J1 HW HB
// Byte 047 :            - Position_1.J1 HW LB
// Byte 048 :            - Position_1.J1 LW HB
// Byte 049 :            - Position_1.J1 LW LB
// Byte 050 : REAL       - Position_1.J2 HW HB
// Byte 051 :            - Position_1.J2 HW LB
// Byte 052 :            - Position_1.J2 LW HB
// Byte 053 :            - Position_1.J2 LW LB
// Byte 054 : REAL       - Position_1.J3 HW HB
// Byte 055 :            - Position_1.J3 HW LB
// Byte 056 :            - Position_1.J3 LW HB
// Byte 057 :            - Position_1.J3 LW LB
// Byte 058 : REAL       - Position_1.J4 HW HB
// Byte 059 :            - Position_1.J4 HW LB
// Byte 060 :            - Position_1.J4 LW HB
// Byte 061 :            - Position_1.J4 LW LB
// Byte 062 : REAL       - Position_1.J5 HW HB
// Byte 063 :            - Position_1.J5 HW LB
// Byte 064 :            - Position_1.J5 LW HB
// Byte 065 :            - Position_1.J5 LW LB
// Byte 066 : REAL       - Position_1.J6 HW HB
// Byte 067 :            - Position_1.J6 HW LB
// Byte 068 :            - Position_1.J6 LW HB
// Byte 069 :            - Position_1.J6 LW LB
// Byte 070 : REAL       - Position_1.E1 HW HB
// Byte 071 :            - Position_1.E1 HW LB
// Byte 072 :            - Position_1.E1 LW HB
// Byte 073 :            - Position_1.E1 LW LB
// Byte 074 : REAL       - Position_2.J1 HW HB
// Byte 075 :            - Position_2.J1 HW LB
// Byte 076 :            - Position_2.J1 LW HB
// Byte 077 :            - Position_2.J1 LW LB
// Byte 078 : REAL       - Position_2.J2 HW HB
// Byte 079 :            - Position_2.J2 HW LB
// Byte 080 :            - Position_2.J2 LW HB
// Byte 081 :            - Position_2.J2 LW LB
// Byte 082 : REAL       - Position_2.J3 HW HB
// Byte 083 :            - Position_2.J3 HW LB
// Byte 084 :            - Position_2.J3 LW HB
// Byte 085 :            - Position_2.J3 LW LB
// Byte 086 : REAL       - Position_2.J4 HW HB
// Byte 087 :            - Position_2.J4 HW LB
// Byte 088 :            - Position_2.J4 LW HB
// Byte 089 :            - Position_2.J4 LW LB
// Byte 090 : REAL       - Position_2.J5 HW HB
// Byte 091 :            - Position_2.J5 HW LB
// Byte 092 :            - Position_2.J5 LW HB
// Byte 093 :            - Position_2.J5 LW LB
// Byte 094 : REAL       - Position_2.J6 HW HB
// Byte 095 :            - Position_2.J6 HW LB
// Byte 096 :            - Position_2.J6 LW HB
// Byte 097 :            - Position_2.J6 LW LB
// Byte 098 : REAL       - Position_2.E1 HW HB
// Byte 099 :            - Position_2.E1 HW LB
// Byte 100 :            - Position_2.E1 LW HB
// Byte 101 :            - Position_2.E1 LW LB
// Byte 102 : REAL       - Position_1.E1 HW HB
// Byte 103 :            - Position_1.E2 HW LB
// Byte 104 :            - Position_1.E2 LW HB
// Byte 105 :            - Position_1.E2 LW LB
// Byte 106 : REAL       - Position_1.E3 HW HB
// Byte 107 :            - Position_1.E3 HW LB
// Byte 108 :            - Position_1.E3 LW HB
// Byte 109 :            - Position_1.E3 LW LB
// Byte 110 : REAL       - Position_1.E4 HW HB
// Byte 111 :            - Position_1.E4 HW LB
// Byte 112 :            - Position_1.E4 LW HB
// Byte 113 :            - Position_1.E4 LW LB
// Byte 114 : REAL       - Position_1.E5 HW HB
// Byte 115 :            - Position_1.E5 HW LB
// Byte 116 :            - Position_1.E5 LW HB
// Byte 117 :            - Position_1.E5 LW LB
// Byte 118 : REAL       - Position_1.E6 HW HB
// Byte 119 :            - Position_1.E6 HW LB
// Byte 120 :            - Position_1.E6 LW HB
// Byte 121 :            - Position_1.E6 LW LB
// Byte 122 : REAL       - Position_2.E2 HW HB
// Byte 123 :            - Position_2.E2 HW LB
// Byte 124 :            - Position_2.E2 LW HB
// Byte 125 :            - Position_2.E2 LW LB
// Byte 125 : REAL       - Position_2.E3 HW HB
// Byte 127 :            - Position_2.E3 HW LB
// Byte 128 :            - Position_2.E3 LW HB
// Byte 129 :            - Position_2.E3 LW LB
// Byte 130 : REAL       - Position_2.E4 HW HB
// Byte 131 :            - Position_2.E4 HW LB
// Byte 132 :            - Position_2.E4 LW HB
// Byte 133 :            - Position_2.E4 LW LB
// Byte 134 : REAL       - Position_2.E5 HW HB
// Byte 135 :            - Position_2.E5 HW LB
// Byte 136 :            - Position_2.E5 LW HB
// Byte 137 :            - Position_2.E5 LW LB
// Byte 138 : REAL       - Position_2.E6 HW HB
// Byte 139 :            - Position_2.E6 HW LB
// Byte 140 :            - Position_2.E6 LW HB
// Byte 141 :            - Position_2.E6 LW LB
// set command parameter 
_command.CmdTyp             :=  CmdType.LoadMeasurementAutomatic;
_command.ExecMode           :=  ExecMode;
_command.ParSeq             := _command.ParSeq;
_command.Priority           :=  Priority;

_command.Mass               := parCmd.Mass;
_command.Mode               := parCmd.Mode;
_command.Reserved           := 0;
_command.Area_J3            := parCmd.Area_J3;
_command.Area_J4            := parCmd.Area_J4;
_command.Area_J5            := parCmd.Area_J5;
_command.Area_J6            := parCmd.Area_J6;
_command.ConfigurationAngle := parCmd.ConfigurationAngle;
_command.Position_1         := parCmd.Position_1;
_command.Position_2         := parCmd.Position_2;


// copy command data to header
_cmdHeader := _command;
// call base implementation to copy header to payload buffer
CreateCommandPayload := SUPER^.CreateCommandPayload(AxesGroup := AxesGroup);

// add command.Mass
CreateCommandPayload.AddReal(_command.Mass);
// add command.Mode
CreateCommandPayload.AddUsint(_command.Mode);
// add command.Reserved
CreateCommandPayload.AddByte(_command.Reserved);
// add command.Area_J3[0]
CreateCommandPayload.AddReal(_command.Area_J3[0]);
// add command.Area_J3[1]
CreateCommandPayload.AddReal(_command.Area_J3[1]);
// add command.Area_J4[0]
CreateCommandPayload.AddReal(_command.Area_J4[0]);
// add command.Area_J4[1]
CreateCommandPayload.AddReal(_command.Area_J4[1]);
// add command.Area_J5[0]
CreateCommandPayload.AddReal(_command.Area_J5[0]);
// add command.Area_J5[1]
CreateCommandPayload.AddReal(_command.Area_J5[1]);
// add command.Area_J6[0]
CreateCommandPayload.AddReal(_command.Area_J6[0]);
// add command.Area_J6[1]
CreateCommandPayload.AddReal(_command.Area_J6[1]);
// add command.ConfigurationAngle
CreateCommandPayload.AddReal(_command.ConfigurationAngle);
// add command.Position_1.J1
CreateCommandPayload.AddReal(_command.Position_1.J1);
// add command.Position_1.J2
CreateCommandPayload.AddReal(_command.Position_1.J2);
// add command.Position_1.J3
CreateCommandPayload.AddReal(_command.Position_1.J3);
// add command.Position_1.J4
CreateCommandPayload.AddReal(_command.Position_1.J4);
// add command.Position_1.J5
CreateCommandPayload.AddReal(_command.Position_1.J5);
// add command.Position_1.J6
CreateCommandPayload.AddReal(_command.Position_1.J6);
// add command.Position_1.E1
CreateCommandPayload.AddReal(_command.Position_1.E1);
// add command.Position_1.E2
CreateCommandPayload.AddReal(_command.Position_1.E2);
// add command.Position_1.E3
CreateCommandPayload.AddReal(_command.Position_1.E3);
// add command.Position_1.E4
CreateCommandPayload.AddReal(_command.Position_1.E4);
// add command.Position_1.E5
CreateCommandPayload.AddReal(_command.Position_1.E5);
// add command.Position_1.E6
CreateCommandPayload.AddReal(_command.Position_1.E6);
// add command.Position_2.J1
CreateCommandPayload.AddReal(_command.Position_2.J1);
// add command.Position_2.J2
CreateCommandPayload.AddReal(_command.Position_2.J2);
// add command.Position_2.J3
CreateCommandPayload.AddReal(_command.Position_2.J3);
// add command.Position_2.J4
CreateCommandPayload.AddReal(_command.Position_2.J4);
// add command.Position_2.J5
CreateCommandPayload.AddReal(_command.Position_2.J5);
// add command.Position_2.J6
CreateCommandPayload.AddReal(_command.Position_2.J6);
// add command.Position_2.E1
CreateCommandPayload.AddReal(_command.Position_2.E1);
// add command.Position_2.E2
CreateCommandPayload.AddReal(_command.Position_2.E2);
// add command.Position_2.E3
CreateCommandPayload.AddReal(_command.Position_2.E3);
// add command.Position_2.E4
CreateCommandPayload.AddReal(_command.Position_2.E4);
// add command.Position_2.E5
CreateCommandPayload.AddReal(_command.Position_2.E5);
// add command.Position_2.E6
CreateCommandPayload.AddReal(_command.Position_2.E6);

// Create logging
CreateCommandPayloadLog(AxesGroup := AxesGroup);
END_METHOD

METHOD INTERNAL CreateCommandPayloadLog 
VAR_IN_OUT
  /// Robot assignment of function
  AxesGroup : AxesGroup; 
END_VAR
// Create log entry for Parameter start
CreateLogMessage      ( Timestamp   := AxesGroup.InternalData.SystemTime,
                        MessageType := MessageType.CMD,
                        Severity    := Severity.DEBUG,
                        MessageCode := 0,
                        MessageText := 'Create command payload with the following parameter(s) :');

// Create log entry for Mass
CreateLogMessagePara1 ( Timestamp   := AxesGroup.InternalData.SystemTime,
                        MessageType := MessageType.CMD,
                        Severity    := Severity.DEBUG,
                        MessageCode := 0,
                        MessageText := 'Command.Mass = {1}',
                        Para1       :=  REAL_TO_STRING(_command.Mass));

// Create log entry for Mode
CreateLogMessagePara1 ( Timestamp   := AxesGroup.InternalData.SystemTime,
                        MessageType := MessageType.CMD,
                        Severity    := Severity.DEBUG,
                        MessageCode := 0,
                        MessageText := 'Command.Mode = {1}',
                        Para1       :=  LOAD_MEASUREMENT_MODE_TO_STRING(_command.Mode));

// Create log entry for Reserved
CreateLogMessagePara1 ( Timestamp   := AxesGroup.InternalData.SystemTime,
                        MessageType := MessageType.CMD,
                        Severity    := Severity.DEBUG,
                        MessageCode := 0,
                        MessageText := 'Command.Reserved = {1}',
                        Para1       :=  REAL_TO_STRING(_command.Reserved));

// Create log entry for Area_J3[0]
CreateLogMessagePara1 ( Timestamp   := AxesGroup.InternalData.SystemTime,
                        MessageType := MessageType.CMD,
                        Severity    := Severity.DEBUG,
                        MessageCode := 0,
                        MessageText := 'Command.Area_J3[0] = {1}',
                        Para1       :=  REAL_TO_STRING(_command.Area_J3[0]));

// Create log entry for Area_J3[1]
CreateLogMessagePara1 ( Timestamp   := AxesGroup.InternalData.SystemTime,
                        MessageType := MessageType.CMD,
                        Severity    := Severity.DEBUG,
                        MessageCode := 0,
                        MessageText := 'Command.Area_J3[1] = {1}',
                        Para1       :=  REAL_TO_STRING(_command.Area_J3[1]));
                        
// Create log entry for Area_J4[0]
CreateLogMessagePara1 ( Timestamp   := AxesGroup.InternalData.SystemTime,
                        MessageType := MessageType.CMD,
                        Severity    := Severity.DEBUG,
                        MessageCode := 0,
                        MessageText := 'Command.Area_J4[0] = {1}',
                        Para1       :=  REAL_TO_STRING(_command.Area_J4[0]));

// Create log entry for Area_J4[1]
CreateLogMessagePara1 ( Timestamp   := AxesGroup.InternalData.SystemTime,
                        MessageType := MessageType.CMD,
                        Severity    := Severity.DEBUG,
                        MessageCode := 0,
                        MessageText := 'Command.Area_J4[1] = {1}',
                        Para1       :=  REAL_TO_STRING(_command.Area_J4[1]));

// Create log entry for Area_J5[0]
CreateLogMessagePara1 ( Timestamp   := AxesGroup.InternalData.SystemTime,
                        MessageType := MessageType.CMD,
                        Severity    := Severity.DEBUG,
                        MessageCode := 0,
                        MessageText := 'Command.Area_J5[0] = {1}',
                        Para1       :=  REAL_TO_STRING(_command.Area_J5[0]));

// Create log entry for Area_J5[1]
CreateLogMessagePara1 ( Timestamp   := AxesGroup.InternalData.SystemTime,
                        MessageType := MessageType.CMD,
                        Severity    := Severity.DEBUG,
                        MessageCode := 0,
                        MessageText := 'Command.Area_J5[1] = {1}',
                        Para1       :=  REAL_TO_STRING(_command.Area_J5[1]));
                        
// Create log entry for Area_J6[0]
CreateLogMessagePara1 ( Timestamp   := AxesGroup.InternalData.SystemTime,
                        MessageType := MessageType.CMD,
                        Severity    := Severity.DEBUG,
                        MessageCode := 0,
                        MessageText := 'Command.Area_J6[0] = {1}',
                        Para1       :=  REAL_TO_STRING(_command.Area_J6[0]));

// Create log entry for Area_J6[1]
CreateLogMessagePara1 ( Timestamp   := AxesGroup.InternalData.SystemTime,
                        MessageType := MessageType.CMD,
                        Severity    := Severity.DEBUG,
                        MessageCode := 0,
                        MessageText := 'Command.Area_J6[1] = {1}',
                        Para1       :=  REAL_TO_STRING(_command.Area_J6[1]));
                        
// Create log entry for ConfigurationAngle
CreateLogMessagePara1 ( Timestamp   := AxesGroup.InternalData.SystemTime,
                        MessageType := MessageType.CMD,
                        Severity    := Severity.DEBUG,
                        MessageCode := 0,
                        MessageText := 'Command.ConfigurationAngle = {1}',
                        Para1       :=  REAL_TO_STRING(_command.ConfigurationAngle));

// Create log entry for Position_1.J1
CreateLogMessagePara1 ( Timestamp   := AxesGroup.InternalData.SystemTime,
                        MessageType := MessageType.CMD,
                        Severity    := Severity.DEBUG,
                        MessageCode := 0,
                        MessageText := 'Command.Position_1.J1 = {1}',
                        Para1       :=  REAL_TO_STRING(_command.Position_1.J1));

// Create log entry for Position_1.J2
CreateLogMessagePara1 ( Timestamp   := AxesGroup.InternalData.SystemTime,
                        MessageType := MessageType.CMD,
                        Severity    := Severity.DEBUG,
                        MessageCode := 0,
                        MessageText := 'Command.Position_1.J2 = {1}',
                        Para1       :=  REAL_TO_STRING(_command.Position_1.J2));
                        
// Create log entry for Position_1.J3
CreateLogMessagePara1 ( Timestamp   := AxesGroup.InternalData.SystemTime,
                        MessageType := MessageType.CMD,
                        Severity    := Severity.DEBUG,
                        MessageCode := 0,
                        MessageText := 'Command.Position_1.J3 = {1}',
                        Para1       :=  REAL_TO_STRING(_command.Position_1.J3));
                        
// Create log entry for Position_1.J4
CreateLogMessagePara1 ( Timestamp   := AxesGroup.InternalData.SystemTime,
                        MessageType := MessageType.CMD,
                        Severity    := Severity.DEBUG,
                        MessageCode := 0,
                        MessageText := 'Command.Position_1.J4 = {1}',
                        Para1       :=  REAL_TO_STRING(_command.Position_1.J4));
                        
// Create log entry for Position_1.J5
CreateLogMessagePara1 ( Timestamp   := AxesGroup.InternalData.SystemTime,
                        MessageType := MessageType.CMD,
                        Severity    := Severity.DEBUG,
                        MessageCode := 0,
                        MessageText := 'Command.Position_1.J5 = {1}',
                        Para1       :=  REAL_TO_STRING(_command.Position_1.J5));

// Create log entry for Position_1.J6
CreateLogMessagePara1 ( Timestamp   := AxesGroup.InternalData.SystemTime,
                        MessageType := MessageType.CMD,
                        Severity    := Severity.DEBUG,
                        MessageCode := 0,
                        MessageText := 'Command.Position_1.J6 = {1}',
                        Para1       :=  REAL_TO_STRING(_command.Position_1.J6));

// Create log entry for Position_1.E1
CreateLogMessagePara1 ( Timestamp   := AxesGroup.InternalData.SystemTime,
                        MessageType := MessageType.CMD,
                        Severity    := Severity.DEBUG,
                        MessageCode := 0,
                        MessageText := 'Command.Position_1.E1 = {1}',
                        Para1       :=  REAL_TO_STRING(_command.Position_1.E1));

// Create log entry for Position_2.J1
CreateLogMessagePara1 ( Timestamp   := AxesGroup.InternalData.SystemTime,
                        MessageType := MessageType.CMD,
                        Severity    := Severity.DEBUG,
                        MessageCode := 0,
                        MessageText := 'Command.Position_2.J1 = {1}',
                        Para1       :=  REAL_TO_STRING(_command.Position_2.J1));

// Create log entry for Position_2.J2
CreateLogMessagePara1 ( Timestamp   := AxesGroup.InternalData.SystemTime,
                        MessageType := MessageType.CMD,
                        Severity    := Severity.DEBUG,
                        MessageCode := 0,
                        MessageText := 'Command.Position_2.J2 = {1}',
                        Para1       :=  REAL_TO_STRING(_command.Position_2.J2));
                        
// Create log entry for Position_2.J3
CreateLogMessagePara1 ( Timestamp   := AxesGroup.InternalData.SystemTime,
                        MessageType := MessageType.CMD,
                        Severity    := Severity.DEBUG,
                        MessageCode := 0,
                        MessageText := 'Command.Position_2.J3 = {1}',
                        Para1       :=  REAL_TO_STRING(_command.Position_2.J3));
                        
// Create log entry for Position_2.J4
CreateLogMessagePara1 ( Timestamp   := AxesGroup.InternalData.SystemTime,
                        MessageType := MessageType.CMD,
                        Severity    := Severity.DEBUG,
                        MessageCode := 0,
                        MessageText := 'Command.Position_2.J4 = {1}',
                        Para1       :=  REAL_TO_STRING(_command.Position_2.J4));
                        
// Create log entry for Position_2.J5
CreateLogMessagePara1 ( Timestamp   := AxesGroup.InternalData.SystemTime,
                        MessageType := MessageType.CMD,
                        Severity    := Severity.DEBUG,
                        MessageCode := 0,
                        MessageText := 'Command.Position_2.J5 = {1}',
                        Para1       :=  REAL_TO_STRING(_command.Position_2.J5));

// Create log entry for Position_2.J6
CreateLogMessagePara1 ( Timestamp   := AxesGroup.InternalData.SystemTime,
                        MessageType := MessageType.CMD,
                        Severity    := Severity.DEBUG,
                        MessageCode := 0,
                        MessageText := 'Command.Position_2.J6 = {1}',
                        Para1       :=  REAL_TO_STRING(_command.Position_2.J6));

// Create log entry for Position_2.E1
CreateLogMessagePara1 ( Timestamp   := AxesGroup.InternalData.SystemTime,
                        MessageType := MessageType.CMD,
                        Severity    := Severity.DEBUG,
                        MessageCode := 0,
                        MessageText := 'Command.Position_2.E1 = {1}',
                        Para1       :=  REAL_TO_STRING(_command.Position_2.E1));
                        
// Create log entry for Position_1.E2
CreateLogMessagePara1 ( Timestamp   := AxesGroup.InternalData.SystemTime,
                        MessageType := MessageType.CMD,
                        Severity    := Severity.DEBUG,
                        MessageCode := 0,
                        MessageText := 'Command.Position_1.E2 = {1}',
                        Para1       :=  REAL_TO_STRING(_command.Position_1.E2));
                        
// Create log entry for Position_1.E3
CreateLogMessagePara1 ( Timestamp   := AxesGroup.InternalData.SystemTime,
                        MessageType := MessageType.CMD,
                        Severity    := Severity.DEBUG,
                        MessageCode := 0,
                        MessageText := 'Command.Position_1.E3 = {1}',
                        Para1       :=  REAL_TO_STRING(_command.Position_1.E3));

// Create log entry for Position_1.E4
CreateLogMessagePara1 ( Timestamp   := AxesGroup.InternalData.SystemTime,
                        MessageType := MessageType.CMD,
                        Severity    := Severity.DEBUG,
                        MessageCode := 0,
                        MessageText := 'Command.Position_1.E4 = {1}',
                        Para1       :=  REAL_TO_STRING(_command.Position_1.E4));
                        
// Create log entry for Position_1.E5
CreateLogMessagePara1 ( Timestamp   := AxesGroup.InternalData.SystemTime,
                        MessageType := MessageType.CMD,
                        Severity    := Severity.DEBUG,
                        MessageCode := 0,
                        MessageText := 'Command.Position_1.E5 = {1}',
                        Para1       :=  REAL_TO_STRING(_command.Position_1.E5));
                        
// Create log entry for Position_1.E6
CreateLogMessagePara1 ( Timestamp   := AxesGroup.InternalData.SystemTime,
                        MessageType := MessageType.CMD,
                        Severity    := Severity.DEBUG,
                        MessageCode := 0,
                        MessageText := 'Command.Position_1.E6 = {1}',
                        Para1       :=  REAL_TO_STRING(_command.Position_1.E6));                

// Create log entry for Position_2.E2
CreateLogMessagePara1 ( Timestamp   := AxesGroup.InternalData.SystemTime,
                        MessageType := MessageType.CMD,
                        Severity    := Severity.DEBUG,
                        MessageCode := 0,
                        MessageText := 'Command.Position_2.E2 = {1}',
                        Para1       :=  REAL_TO_STRING(_command.Position_2.E2));
                        
// Create log entry for Position_2.E3
CreateLogMessagePara1 ( Timestamp   := AxesGroup.InternalData.SystemTime,
                        MessageType := MessageType.CMD,
                        Severity    := Severity.DEBUG,
                        MessageCode := 0,
                        MessageText := 'Command.Position_2.E3 = {1}',
                        Para1       :=  REAL_TO_STRING(_command.Position_2.E3));

// Create log entry for Position_2.E4
CreateLogMessagePara1 ( Timestamp   := AxesGroup.InternalData.SystemTime,
                        MessageType := MessageType.CMD,
                        Severity    := Severity.DEBUG,
                        MessageCode := 0,
                        MessageText := 'Command.Position_2.E4 = {1}',
                        Para1       :=  REAL_TO_STRING(_command.Position_2.E4));
                        
// Create log entry for Position_2.E5
CreateLogMessagePara1 ( Timestamp   := AxesGroup.InternalData.SystemTime,
                        MessageType := MessageType.CMD,
                        Severity    := Severity.DEBUG,
                        MessageCode := 0,
                        MessageText := 'Command.Position_2.E5 = {1}',
                        Para1       :=  REAL_TO_STRING(_command.Position_2.E5));
                        
// Create log entry for Position_2.E6
CreateLogMessagePara1 ( Timestamp   := AxesGroup.InternalData.SystemTime,
                        MessageType := MessageType.CMD,
                        Severity    := Severity.DEBUG,
                        MessageCode := 0,
                        MessageText := 'Command.Position_2.E6 = {1}',
                        Para1       :=  REAL_TO_STRING(_command.Position_2.E6));
END_METHOD

METHOD FB_init : BOOL
VAR_INPUT
  /// if TRUE, the retain variables are initialized (warm start / cold start)
  bInitRetains : BOOL; 
  /// if TRUE, the instance afterwards gets moved into the copy code (online change)
  bInCopyCode  : BOOL;  
END_VAR
MyType := 'MC_LoadMeasurementAutomaticFB';
END_METHOD

METHOD PROTECTED OnCall
VAR_IN_OUT
  /// Robot assignment of function
  AxesGroup : AxesGroup; 
END_VAR
// call base implementation
SUPER^.OnCall(AxesGroup := AxesGroup);

CASE _stepCmd OF
  
  00:  IF ( _execute_R.Q )  
       THEN
         // Check function is supported and parameter are valid ?
         IF (( CheckFunctionSupported( AxesGroup := AxesGroup )) AND
             ( CheckParameterValid   ( AxesGroup := AxesGroup )))      
         THEN
           // set busy flag
           Busy := TRUE;
           // Reset command outputs
           SysDepMemSet(pDest := ADR(OutCmd), Value := 0, DataLen := SIZEOF(OutCmd));         
           // apply command parameter
          _parCmd := ParCmd;
           // init parameter sequence
          _command.ParSeq := 1;
           // create command data
           CommandData := CreateCommandPayload(AxesGroup := AxesGroup);
           // Add command to active command register
          _uniqueID := AxesGroup.Acyclic.ActiveCommandRegister.AddCmd( pCommandFB := ADR(THIS^ ));     
           // set timeout
           SetTimeout(PT := _timeoutCmd, rTimer := _timerCmd);
           // inc step counter
          _stepCmd := _stepCmd + 1;
         END_IF 
       END_IF
     

  01:  // Wait for responce received
       IF ( _responseReceived )
       THEN
         // reset response received flag
        _responseReceived := FALSE;
         // reset Active flag
         Active := FALSE;
         
         CASE  _response.State 
         OF
           CmdMessageState.BUFFERED    : CommandBuffered    := TRUE;
           CmdMessageState.ACTIVE      : Active             := TRUE;
           CmdMessageState.INTERRUPTED : CommandInterrupted := TRUE;
           CmdMessageState.DONE        : Done               := TRUE;
           CmdMessageState.ABORTED     : CommandAborted     := TRUE;
           CmdMessageState.ERROR       : Error              := TRUE;
         END_CASE
                
         // Done, Aborted or Error ?
         IF (_response.State >= CmdMessageState.DONE )
         THEN
           // Reset Busy flag
           Busy := FALSE;     
           // Update results
           OutCmd.LoadData          := _response.LoadData;
           OutCmd.LoadDataAvailable := _response.LoadDataAvailable;
           // set timeout
           SetTimeout(PT := _timeoutCmd, rTimer := _timerCmd);
           // inc step counter
          _stepCmd := _stepCmd + 1; 
         END_IF
       END_IF


  02: IF ( NOT Execute)
      THEN
        Reset();
      END_IF     
      
ELSE
  // invalid step
  ErrorID := RobotLibraryEvents.ERR_INVALID_STEP;
END_CASE


// Reset FB
IF ( NOT Execute )
THEN
  Reset();
END_IF
END_METHOD

METHOD INTERNAL ParseResponsePayload : DINT
VAR_INPUT
  /// Response data
  ResponseData : RobotLibraryRecvDataFB;
  /// Timestamp
  Timestamp    : SystemTime;  
END_VAR
// Table 6-778: Sent CMD payload (PLC to RC) of "LoadMeasurementAutomatic"
// --------------------------
// Header
// --------------------------
// Byte 00 : USINT - ParSeq | State     
// Byte 01 : SINT  - AlarmMessageSeverity    
// Byte 02 : UINT  - AlarmMessageCode HB
// Byte 03 :       - AlarmMessageCode LB
// Datablock
// --------------------------
// Byte 004 : IEC_DATE   - IEC Date LW HB
// Byte 005 :            - IEC Date LW LB
// Byte 006 : IEC_TIME   - IEC Time HW HB
// Byte 007 :            - IEC Time HW LB
// Byte 008 :            - IEC Time LW HB
// Byte 009 :            - IEC Time LW LB
// Byte 010 : REAL       - LoadData.X HW HB
// Byte 011 :            - LoadData.X HW LB
// Byte 012 :            - LoadData.X LW HB
// Byte 013 :            - LoadData.X LW LB
// Byte 014 : REAL       - LoadData.Y HW HB
// Byte 015 :            - LoadData.Y HW LB
// Byte 016 :            - LoadData.Y LW HB
// Byte 017 :            - LoadData.Y LW LB
// Byte 018 : REAL       - LoadData.Z HW HB
// Byte 019 :            - LoadData.Z HW LB
// Byte 020 :            - LoadData.Z LW HB
// Byte 021 :            - LoadData.Z LW LB
// Byte 022 : REAL       - LoadData.Rx HW HB
// Byte 023 :            - LoadData.Rx HW LB
// Byte 024 :            - LoadData.Rx LW HB
// Byte 025 :            - LoadData.Rx LW LB
// Byte 026 : REAL       - LoadData.Ry HW HB
// Byte 027 :            - LoadData.Ry HW LB
// Byte 028 :            - LoadData.Ry LW HB
// Byte 029 :            - LoadData.Ry LW LB
// Byte 030 : REAL       - LoadData.Rz HW HB
// Byte 031 :            - LoadData.Rz HW LB
// Byte 032 :            - LoadData.Rz LW HB
// Byte 033 :            - LoadData.Rz LW LB
// Byte 034 : REAL       - Mass HW HB
// Byte 035 :            - Mass HW LB
// Byte 036 :            - Mass LW HB
// Byte 037 :            - Mass LW LB
// Byte 038 : REAL       - LoadData.Ix HW HB
// Byte 039 :            - LoadData.Ix HW LB
// Byte 040 :            - LoadData.Ix LW HB
// Byte 041 :            - LoadData.Ix LW LB
// Byte 042 : REAL       - LoadData.Iy HW HB
// Byte 043 :            - LoadData.Iy HW LB
// Byte 044 :            - LoadData.Iy LW HB
// Byte 045 :            - LoadData.Iy LW LB
// Byte 046 : REAL       - LoadData.Iz HW HB
// Byte 047 :            - LoadData.Iz HW LB
// Byte 048 :            - LoadData.Iz LW HB
// Byte 049 :            - LoadData.Iz LW LB
// Byte 050 : BOOL       - LoadData.Available
// call base implementation to parse the header from payload buffer
ResponseData.PayloadPtr := SUPER^.ParseResponsePayload(ResponseData := ResponseData, Timestamp := Timestamp);

// copy parsed header to response
_response.ParSeq               := _rspHeader.ParSeq;
_response.State                := _rspHeader.State;
_response.AlarmMessageSeverity := _rspHeader.AlarmMessageSeverity;
_response.AlarmMessageCode     := _rspHeader.AlarmMessageCode;

// Get Response.LoadData.Timestamp.TsData
_response.LoadData.Timestamp.IEC_DATE := ResponseData.GetIecDate();
// Get Response.LoadData.Timestamp.TsTime
_response.LoadData.Timestamp.IEC_TIME := ResponseData.GetIecTime();
// Get Response.LoadData.X
_response.LoadData.X := ResponseData.GetReal();
// Get Response.LoadData.Y
_response.LoadData.Y := ResponseData.GetReal();
// Get Response.LoadData.Z
_response.LoadData.Z := ResponseData.GetReal();
// Get Response.LoadData.Rx
_response.LoadData.Rx := ResponseData.GetReal();
// Get Response.LoadData.Ry
_response.LoadData.Ry := ResponseData.GetReal();
// Get Response.LoadData.Rz
_response.LoadData.Rz := ResponseData.GetReal();
// Get Response.LoadData.Mass
_response.LoadData.Mass := ResponseData.GetReal();
// Get Response.LoadData.Ix
_response.LoadData.Ix := ResponseData.GetReal();
// Get Response.LoadData.Iy
_response.LoadData.Iy := ResponseData.GetReal();
// Get Response.LoadData.Iz
_response.LoadData.Iz := ResponseData.GetReal();
// Get Response.LoadDataAvailable
_response.LoadDataAvailable := ResponseData.GetBool();

// Create logging
ParseResponsePayloadLog(ResponseData := ResponseData, Timestamp := Timestamp);
END_METHOD

METHOD INTERNAL ParseResponsePayloadLog
VAR_INPUT
  /// Response data
  ResponseData : RobotLibraryRecvDataFB;
  /// Timestamp
  Timestamp    : SystemTime;  
END_VAR
// Create log entry for Parameter start
CreateLogMessage      ( Timestamp   := Timestamp,
                        MessageType := MessageType.CMD,
                        Severity    := Severity.DEBUG,
                        MessageCode := 0,
                        MessageText := 'Parsed the following parameter(s) from response data:');
                        
// Create log entry for LoadData.Timestamp.IEC_DATE
CreateLogMessagePara1 ( Timestamp   := Timestamp,
                        MessageType := MessageType.CMD,
                        Severity    := Severity.DEBUG,
                        MessageCode := 0,
                        MessageText := 'Response.LoadData.Timestamp.IEC_DATE = {1}',
                        Para1       :=  IEC_DATE_TO_STRING(_response.LoadData.Timestamp.IEC_DATE));

// Create log entry for LoadData.Timestamp.IEC_TIME
CreateLogMessagePara1 ( Timestamp   := Timestamp,
                        MessageType := MessageType.CMD,
                        Severity    := Severity.DEBUG,
                        MessageCode := 0,
                        MessageText := 'Response.LoadData.Timestamp.IEC_TIME = {1}',
                        Para1       :=  IEC_TIME_TO_STRING(_response.LoadData.Timestamp.IEC_TIME));

// Create log entry for LoadData.X
CreateLogMessagePara1 ( Timestamp   := Timestamp,
                        MessageType := MessageType.CMD,
                        Severity    := Severity.DEBUG,
                        MessageCode := 0,
                        MessageText := 'Response.LoadData.X = {1}',
                        Para1       :=  REAL_TO_STRING(_response.LoadData.X));

// Create log entry for LoadData.Y
CreateLogMessagePara1 ( Timestamp   := Timestamp,
                        MessageType := MessageType.CMD,
                        Severity    := Severity.DEBUG,
                        MessageCode := 0,
                        MessageText := 'Response.LoadData.Y = {1}',
                        Para1       :=  REAL_TO_STRING(_response.LoadData.Y));

// Create log entry for LoadData.Z
CreateLogMessagePara1 ( Timestamp   := Timestamp,
                        MessageType := MessageType.CMD,
                        Severity    := Severity.DEBUG,
                        MessageCode := 0,
                        MessageText := 'Response.LoadData.Z = {1}',
                        Para1       :=  REAL_TO_STRING(_response.LoadData.Z));

// Create log entry for LoadData.Rx
CreateLogMessagePara1 ( Timestamp   := Timestamp,
                        MessageType := MessageType.CMD,
                        Severity    := Severity.DEBUG,
                        MessageCode := 0,
                        MessageText := 'Response.LoadData.Rx = {1}',
                        Para1       :=  REAL_TO_STRING(_response.LoadData.Rx));

// Create log entry for LoadData.Ry
CreateLogMessagePara1 ( Timestamp   := Timestamp,
                        MessageType := MessageType.CMD,
                        Severity    := Severity.DEBUG,
                        MessageCode := 0,
                        MessageText := 'Response.LoadData.Ry = {1}',
                        Para1       :=  REAL_TO_STRING(_response.LoadData.Ry));

// Create log entry for LoadData.Rz
CreateLogMessagePara1 ( Timestamp   := Timestamp,
                        MessageType := MessageType.CMD,
                        Severity    := Severity.DEBUG,
                        MessageCode := 0,
                        MessageText := 'Response.LoadData.Rz = {1}',
                        Para1       :=  REAL_TO_STRING(_response.LoadData.Rz));

// Create log entry for LoadData.Mass
CreateLogMessagePara1 ( Timestamp   := Timestamp,
                        MessageType := MessageType.CMD,
                        Severity    := Severity.DEBUG,
                        MessageCode := 0,
                        MessageText := 'Response.LoadData.Mass = {1}',
                        Para1       :=  REAL_TO_STRING(_response.LoadData.Mass));

// Create log entry for LoadData.Ix
CreateLogMessagePara1 ( Timestamp   := Timestamp,
                        MessageType := MessageType.CMD,
                        Severity    := Severity.DEBUG,
                        MessageCode := 0,
                        MessageText := 'Response.LoadData.Ix = {1}',
                        Para1       :=  REAL_TO_STRING(_response.LoadData.Ix));

// Create log entry for LoadData.Iy
CreateLogMessagePara1 ( Timestamp   := Timestamp,
                        MessageType := MessageType.CMD,
                        Severity    := Severity.DEBUG,
                        MessageCode := 0,
                        MessageText := 'Response.LoadData.Iy = {1}',
                        Para1       :=  REAL_TO_STRING(_response.LoadData.Iy));

// Create log entry for LoadData.Iz
CreateLogMessagePara1 ( Timestamp   := Timestamp,
                        MessageType := MessageType.CMD,
                        Severity    := Severity.DEBUG,
                        MessageCode := 0,
                        MessageText := 'Response.LoadData.Iz = {1}',
                        Para1       :=  REAL_TO_STRING(_response.LoadData.Iz));

// Create log entry for LoadDataAvailable
CreateLogMessagePara1 ( Timestamp   := Timestamp,
                        MessageType := MessageType.CMD,
                        Severity    := Severity.DEBUG,
                        MessageCode := 0,
                        MessageText := 'Response.LoadDataAvailable = {1}',
                        Para1       :=  BOOL_TO_STRING(_response.LoadDataAvailable));
END_METHOD

METHOD PROTECTED Reset : DINT
VAR_INPUT
END_VAR
Reset := SUPER^.Reset();

Done               := FALSE;
Busy               := FALSE;
Active             := FALSE;
CommandBuffered    := FALSE;
CommandAborted     := FALSE;
CommandInterrupted := FALSE;
END_METHOD

END_FUNCTION_BLOCK

// Library/POUs/Calculation/MC_LoadMeasurementSequential/MC_LoadMeasurementSequentialFB
/// Sequential detection of load data
FUNCTION_BLOCK MC_LoadMeasurementSequentialFB EXTENDS RobotLibraryBaseExecuteFB
// ------------------------------------------------------------------------- 
//  SRCI Robot Library                                                
// ------------------------------------------------------------------------- 
//                                                                           
//  Object:      LoadMeasurementSequentialFB                                       
//  Author:      Thorsten Brach                                                
//  Date:        2024-06-01
//
//  Description:                                              
//   
//                                                                           
//  Copyright: 
//    (C) 2024 Thorsten Brach. All rights reserved                                                                                                                                            
//             Licensed under the LGPL-3.0 license.
//                                                                           
//  Disclaimer:                                                                           
//    This project is provided without any guarantee and can be used for   
//    private and commercial purposes. Any use is at the user’s 
//    own risk and responsibility.
//
// -------------------------------------------------------------------------
VAR_INPUT
  /// Processing mode
  ProcessingMode     : ProcessingMode;
  /// Defines the target sequence in which the command will be executed
  SequenceFlag       : SequenceFlag;  
  /// Command parameter 
  ParCmd             : LoadMeasurementSequentialParCmd;      
END_VAR

VAR_OUTPUT
  /// Command is transferred and confirmed by the RC
  CommandBuffered    : BOOL;  
  /// The command takes control of the motion of the according axis group.
  Active             : BOOL;
  /// The command was aborted by another command.
  CommandAborted     : BOOL;
  /// TRUE, while command is interrupted during execution and can be continued.
  CommandInterrupted : BOOL;
  /// Command output 
  OutCmd             : LoadMeasurementSequentialOutCmd;        
END_VAR

VAR
  /// internal copy of command parameter 
 _parCmd             : LoadMeasurementSequentialParCmd;
  /// command data to send
 _command            : LoadMeasurementSequentialSendData;
  /// response data received
 _response           : LoadMeasurementSequentialRecvData;      
END_VAR

SUPER^(AxesGroup := AxesGroup);

METHOD PROTECTED CheckFunctionSupported : BOOL
VAR_IN_OUT
  /// Robot assignment of function
  AxesGroup : AxesGroup; 
END_VAR
CheckFunctionSupported := AxesGroup.InternalData.RCSupportedFunctions.LoadMeasurementSequential;

IF ( NOT CheckFunctionSupported )
THEN
  // call base implementation for set error and create log entry
  SUPER^.CheckFunctionSupported(AxesGroup := AxesGroup);
END_IF
END_METHOD

METHOD PROTECTED CheckParameterChanged : BOOL
VAR_IN_OUT
  /// Robot assignment of function
  AxesGroup    : AxesGroup; 
END_VAR
// Check ParCmd Size is > 0, because MemCmp does not work correctly with size = 0
IF (SIZEOF(ParCmd) = 0) 
THEN 
  RETURN;
END_IF

// compare memory 
_parameterChanged := ( SysDepMemCmp(pData1 := ADR(ParCmd), pData2 := ADR(_parCmd), DataLen := SIZEOF(ParCmd)) <> RobotLibraryConstants.OK );

// check parameter valid ?
_parameterValid   := CheckParameterValid( AxesGroup := AxesGroup );

IF ((  _parameterChanged        )  AND 
    (  _parameterValid          )) OR
    (  _parameterUpdateInternal )  
THEN  
  // reset internal flag for send parameter update
 _parameterUpdateInternal := FALSE;
  // update internal copy of parameters 
 _parCmd := ParCmd;
  // inc parameter sequence
 _command.ParSeq := _command.ParSeq + 1;
  // update command data  
  CommandData := CreateCommandPayload(AxesGroup := AxesGroup); // ( Access via reference to rCommandFB in ACR )
  // notify active command register 
  AxesGroup.Acyclic.ActiveCommandRegister.NotifyParameterChanged := _uniqueID;
END_IF
END_METHOD

METHOD INTERNAL CreateCommandPayload : RobotLibrarySendDataFB
VAR_IN_OUT
  /// Robot assignment of function
  AxesGroup : AxesGroup; 
END_VAR
// Table 6-784: Sent CMD payload (PLC to RC) of "LoadMeasurementSequential"
// --------------------------
// Header
// --------------------------
// Byte 000 : UINT  - Type HB     
// Byte 001 :       - Type LB    
// Byte 002 : USINT - Reserve | ExecutionMode
// Byte 003 : USINT - ParSeq  | Priority
// --------------------------
// Datablock
// --------------------------
// Byte 004 : REAL       - Mass HW HB
// Byte 005 :            - Mass HW LB
// Byte 006 :            - Mass LW HB
// Byte 007 :            - Mass LW LB
// Byte 008 : USINT      - Mode
// set command parameter 
_command.CmdTyp   :=  CmdType.LoadMeasurementSequential;
_command.ExecMode :=  ExecMode;
_command.ParSeq   := _command.ParSeq;
_command.Priority :=  Priority;                  
_command.Mass     :=  parCmd.Mass;
_command.Mode     :=  parCmd.Mode;


// copy command data to header
_cmdHeader := _command;
// call base implementation to copy header to payload buffer
CreateCommandPayload := SUPER^.CreateCommandPayload(AxesGroup := AxesGroup);


// add command.Mass
CreateCommandPayload.AddReal(_command.Mass);
// add command.Mode
CreateCommandPayload.AddUsint(_command.Mode);

// Create logging
CreateCommandPayloadLog(AxesGroup := AxesGroup);
END_METHOD

METHOD INTERNAL CreateCommandPayloadLog 
VAR_IN_OUT
  /// Robot assignment of function
  AxesGroup : AxesGroup; 
END_VAR
// Create log entry for Parameter start
CreateLogMessage      ( Timestamp   := AxesGroup.InternalData.SystemTime,
                        MessageType := MessageType.CMD,
                        Severity    := Severity.DEBUG,
                        MessageCode := 0,
                        MessageText := 'Create command payload with the following parameter(s) :');

// Create log entry for Mass
CreateLogMessagePara1 ( Timestamp   := AxesGroup.InternalData.SystemTime,
                        MessageType := MessageType.CMD,
                        Severity    := Severity.DEBUG,
                        MessageCode := 0,
                        MessageText := 'Command.Mass = {1}',
                        Para1       :=  REAL_TO_STRING(_command.Mass));
                        
// Create log entry for Mode
CreateLogMessagePara1 ( Timestamp   := AxesGroup.InternalData.SystemTime,
                        MessageType := MessageType.CMD,
                        Severity    := Severity.DEBUG,
                        MessageCode := 0,
                        MessageText := 'Command.Mode = {1}',
                        Para1       :=  LOAD_MEASUREMENT_STEPS_TO_STRING(_command.Mode));
END_METHOD

METHOD FB_init : BOOL
VAR_INPUT
  /// if TRUE, the retain variables are initialized (warm start / cold start)
  bInitRetains : BOOL; 
  /// if TRUE, the instance afterwards gets moved into the copy code (online change)
  bInCopyCode  : BOOL;  
END_VAR
MyType := 'MC_LoadMeasurementSequentialFB';

ExecMode := ExecutionMode.PARALLEL;
END_METHOD

METHOD PROTECTED OnCall
VAR_IN_OUT
  /// Robot assignment of function
  AxesGroup : AxesGroup; 
END_VAR
// call base implementation
SUPER^.OnCall(AxesGroup := AxesGroup);

CASE _stepCmd OF
  
  00:  IF ( _execute_R.Q ) 
       THEN
         // Check function is supported and parameter are valid ?
         IF (( CheckFunctionSupported( AxesGroup := AxesGroup )) AND
             ( CheckParameterValid   ( AxesGroup := AxesGroup )))      
         THEN
           // set busy flag
           Busy := TRUE;
           // Reset command outputs
           SysDepMemSet(pDest := ADR(OutCmd), Value := 0, DataLen := SIZEOF(OutCmd));         
           // apply command parameter
          _parCmd := ParCmd;
           // init parameter sequence
          _command.ParSeq := 1;
           // create command data
           CommandData := CreateCommandPayload(AxesGroup := AxesGroup);
           // Add command to active command register
          _uniqueID := AxesGroup.Acyclic.ActiveCommandRegister.AddCmd( pCommandFB := ADR(THIS^ ));     
           // set timeout
           SetTimeout(PT := _timeoutCmd, rTimer := _timerCmd);
           // inc step counter
          _stepCmd := _stepCmd + 1; 
         END_IF
       END_IF
     

  01:  // Wait for responce received
       IF ( _responseReceived )
       THEN
         // reset response received flag
        _responseReceived := FALSE;
         // reset Active flag
         Active := FALSE;
         
         CASE  _response.State 
         OF
           CmdMessageState.ACTIVE      : Active             := TRUE;
           CmdMessageState.BUFFERED    : CommandBuffered    := TRUE;
           CmdMessageState.INTERRUPTED : CommandInterrupted := TRUE;
           CmdMessageState.DONE        : Done               := TRUE;
           CmdMessageState.ABORTED     : CommandAborted     := TRUE;
           CmdMessageState.ERROR       : Error              := TRUE;
         END_CASE
                
